{attribute 'linkalways'} 
{attribute 'no_explicit_call' := 'This FB is a CLASS and must be accessed using methods or properties'}
{attribute 'enable_dynamic_creation'}
FUNCTION_BLOCK Node_F_VN_ClipLineToBoundary_ITcVnImage EXTENDS VisionNode
VAR
    aLine : _TcVnVector4_LREAL;
    ipImage : _ITcVnImage;
    aStartPoint : _TcVnPoint2_REAL;
    aEndPoint : _TcVnPoint2_REAL;
    hrPrev : _HRESULT(S_OK);
	hresult : _HRESULT(S_OK);
END_VAR

METHOD PUBLIC  Clone : I_Node
VAR
	pNode : POINTER TO Node_F_VN_ClipLineToBoundary_ITcVnImage;
END_VAR
pNode := __NEW(Node_F_VN_ClipLineToBoundary_ITcVnImage);
Clone := pNode^;
END_METHOD

METHOD FB_init : BOOL
VAR_INPUT
	bInitRetains : BOOL; // if TRUE, the retain variables are initialized (warm start / cold start)
	bInCopyCode : BOOL;  // if TRUE, the instance afterwards gets moved into the copy code (online change)
END_VAR
AddInput('aLine', aLine);
AddInput('ipImage', ipImage);
AddInput('aStartPoint', aStartPoint);
AddInput('aEndPoint', aEndPoint);
AddInput('hrPrev', hrPrev);
AddOutput('aLine', aLine);
AddOutput('aStartPoint', aStartPoint);
AddOutput('aEndPoint', aEndPoint);
AddOutput('hresult',hresult);
END_METHOD

METHOD PROTECTED OnExecute
hresult.Value := F_VN_ClipLineToBoundary_ITcVnImage(
	aLine := aLine.Value,
    ipImage := ipImage.Value,
    aStartPoint := aStartPoint.Value,
    aEndPoint := aEndPoint.Value,
	hrPrev:= hrPrev.Value);
END_METHOD

METHOD PUBLIC PreExecutionCheck
VAR_INPUT
	Check : I_PreExecutionChecks;
END_VAR
Check.IsTrue(ipImage.IsValid, 'ipImage must contain an image');
END_METHOD

END_FUNCTION_BLOCK

(* stored: Version 1.1.0.1, ProductVersion 3.1.4024.13
   POU Node_F_VN_ClipLineToBoundary_ITcVnImage: Id {8d588fac-f33b-0da8-1d26-f320a070bbf6}, SpecialFunc None
   Folder Constructor: Id {09ef37e3-ca25-09af-1285-041a1412b990}
   Method Clone: Id {33c8fd8f-db59-0555-2aaa-31cfa3499fbf}
   Method FB_init: Id {9e5995cf-c307-05c8-0107-f1508a370369}
   Method OnExecute: Id {f1d95874-41c8-07ee-29a9-d0d3e857e103}
   Method PreExecutionCheck: Id {bb946d39-3d88-0b1e-1b44-8929eb854957} *)
